PROGRAM MAIN
VAR
	bTemp : BOOL;
END_VAR

P_Filtering();
P_Inputs();
P_Output();

END_PROGRAM

(* stored: Version 1.1.0.1
   POU MAIN: Id {73114a79-e8e7-4c77-9271-864ce29939b0}, SpecialFunc None *)
